(* IEC 61131-3 sources: Everest-Indoor-Unit/SWNOVHIDUOUCR00/SWNOVHIDUOUCR00/Sources/Functions/GeneralMng, 3 files *)

(* ---- FindTimezoneIndex.st ---- *)
USING System;
USING System.Timer;

FUNCTION FindTimezoneIndex : UINT
    VAR_IN_OUT CONSTANT
		(**List of time zones available from the software*)
        TimeZonePosixList : ARRAY[*] OF STRING;
		(**The time zone posix to find*)
		TimeZonePosix : STRING;
	END_VAR
    VAR
        i : DINT;
    END_VAR

    FOR i := LOWER_BOUND(TimeZonePosixList, 1) TO UPPER_BOUND(TimeZonePosixList, 1) DO
        IF TimeZonePosix = TimeZonePosixList[i] THEN
            FindTimezoneIndex := TO_UINT(i);
            EXIT;
        END_IF;
    END_FOR;
END_FUNCTION

(* ---- SplitPrjGUID.st ---- *)
USING System;
USING System.Text;
USING System.Timer;
USING System.Serial;
USING System.Math;

(**Returns Stone project GUID splitted.*)
FUNCTION SplitPrjGUID : StonePrjGUID
    VAR_IN_OUT CONSTANT
        (**↓ Stone project GUID*)
        ProjectID : STRING;
    END_VAR
    SplitPrjGUID.Grp1 := MID(ProjectID,  8, 1);
    SplitPrjGUID.Grp2 := MID(ProjectID,  4, 1+8);
    SplitPrjGUID.Grp3 := MID(ProjectID,  4, 1+8+4);
    SplitPrjGUID.Grp4 := MID(ProjectID,  4, 1+8+4+4);
    SplitPrjGUID.Grp5 := MID(ProjectID, 12, 1+8+4+4+4);
END_FUNCTION

(* ---- SoftwareSafeUpload.st ---- *)
USING System;
USING System.Timer;

(**
 * Allow to upload the software safely.
 * When a full download request from the IDE starts, the variable "KeybOffOn" will be set to FALSE.
 * Then after 10s, if the StartUpload is TRUE the download will start.
 *)
FUNCTION_BLOCK SoftwareSafeUpload
    VAR_IN_OUT
        (**Keyboard On/Off*)
        KeybOffOn   : BOOL;
    END_VAR
    VAR_INPUT
        (**Upload start-up command*)
        StartUpload : BOOL;
    END_VAR
    VAR
        (**Wait before start software upload inside controller*)
        TON_WAIT_DOWNLOAD : TON := (PT := T#5s);
    END_VAR

    (* A write operation in RETAIN/PERSISTENT MEMORY (ie: KeybOnOff=FALSE) became effective after 5s -> Inside the POP-UP window ->
           if you select button "BY-PASS" (... and NOT WAIT 10s) and the UNIT is ON -> at controller re-start probably KeybOnOff will be TRUE. *)
    TON_WAIT_DOWNLOAD(IN := NOT(KeybOffOn) AND StartUpload);

    IF GetFullDownloadRequest() THEN
        //Request to put in "safety status" the unit.
        KeybOffOn := FALSE;
        //When UNIT is in "safety status", the full download can be done.
        IF TON_WAIT_DOWNLOAD.Q THEN
            SetIDESema(TO_INT(IDESEMA_FULLDOWNLOAD), TO_INT(SEMA_STATUS_GO));
        END_IF;
    ELSE
        SetIDESema(TO_INT(IDESEMA_FULLDOWNLOAD), TO_INT(SEMA_STATUS_WAIT));
    END_IF;
END_FUNCTION_BLOCK
